(* CoDeSys 2.3 export: CHECKDIVREAL.EXP *)

(* POU CheckDivReal, ST *)
FUNCTION CheckDivReal : REAL
VAR_INPUT
	divisor: REAL;
END_VAR
VAR
END_VAR
(* @TEXT_IMPLEMENTATION := 'ST' *)
IF divisor = 0 THEN
	CheckDivReal := 1;
ELSE
	CheckDivReal := divisor;
END_IF
END_FUNCTION
